(* PLC project Tc3_EventLogger.FB_RequestEventDetails Demo, tc3-libraries-kb TwinCAT 3.1 *)
(* stored: creationDateTime 2026-05-11T01:00:00, modificationDateTime 2026-05-11T01:00:00 *)

PROGRAM P_Demo_FB_RequestEventDetails
  VAR
    fbFB_RequestEventDetails : FB_RequestEventDetails;  (* Tc3_EventLogger.FB_RequestEventDetails 实例 *)
    arg_nIndex : UDINT;  (* VAR_INPUT nIndex *)
    arg_fbDetail : REFERENCE TO FB_TcDetail;  (* VAR_INPUT fbDetail *)
    arg_eventClass : GUID;  (* VAR_INPUT eventClass *)
    arg_nEventId : UDINT;  (* VAR_INPUT nEventId *)
    arg_nLangId : DINT;  (* VAR_INPUT nLangId *)
    arg_ipRemoteLogger : I_TcRemoteEventLogger;  (* VAR_INPUT ipRemoteLogger *)
  END_VAR

            // ============================================================
// Tc3_EventLogger.FB_RequestEventDetails 演示程序（FB 实例）
// ============================================================
// 验证步骤：
//   1. 引用 Tc3_EventLogger（及依赖类型所在库 Tc2_System 等）
//   2. 编译 + 登录
//   3. 按 doc.md 给 arg_* 赋值
//   4. 在线监视 out_* / io_* 输出
// ============================================================

fbFB_RequestEventDetails(
    nIndex := arg_nIndex,
    fbDetail := arg_fbDetail,
    eventClass := arg_eventClass,
    nEventId := arg_nEventId,
    nLangId := arg_nLangId,
    ipRemoteLogger := arg_ipRemoteLogger
);

          
END_PROGRAM
